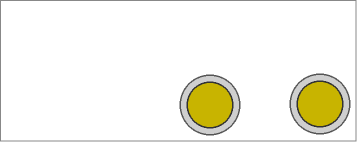
VISUALIZATION Visualization  // 357x142
    Lamp1 (175,70 70x70), variable: GVL1.Lichten, style: Lamp-Lamp1-Yellow
    Lamp1 (285,69 70x70), variable: GVL1.Projectorscherm, style: Lamp-Lamp1-Yellow
END_VISUALIZATION

(* stored: Version 1.1.0.1, ProductVersion 3.1.4022.9
   Visu Visualization: Id {8a15400c-277f-4c6e-aa9a-e38930a493bf} *)
